(* IEC 61131-3 sources: ST-to-Python-Transpiler/AS Projekti/RampController/Program, 3 files *)

(* ---- Types.typ ---- *)
TYPE

END_TYPE

(* ---- Ramp.st ---- *)
PROGRAM _INIT
	(* Insert code here *)

END_PROGRAM

PROGRAM _CYCLIC
	(** --- RAMP CONTROLLER LOGIC --- **)
	Ramp(TARGET := UserSetpoint, CURRENT := CurrentValue, RAMP_UP := RampRateUp, RAMP_DOWN := RampRateDown, ENABLE := RampEnable, RESET := RampReset);
	SmoothSetpoint := Ramp.OUT;
	AtTarget := Ramp.REACHED;

	(** --- DEADBAND FILTER LOGIC --- **)
	Filter(IN := SensorRaw, DEADBAND := Deadband, CENTER := SmoothSetpoint);
	SensorFiltered := Filter.OUT;
	SensorActive := Filter.IS_ACTIVE;

END_PROGRAM

PROGRAM _EXIT
	(* Insert code here *)

END_PROGRAM

(* ---- Variables.var ---- *)
VAR
	UserSetpoint : REAL := 100.0;
	SensorRaw : REAL := 99.7;
	Ramp : RampController;
	Filter : DeadbandFilter; (** Control ramp behavior **)
	RampEnable : BOOL := TRUE;
	RampReset : BOOL := FALSE;
	RampRateUp : REAL := 1.0;
	RampRateDown : REAL := 2.0;
	CurrentValue : REAL := 90.0; (** Parameters for deadband filter **)
	Deadband : REAL := 0.5; (** Output: Ramped setpoint **)
	SmoothSetpoint : REAL; (** Output: Filtered sensor signal **)
	SensorFiltered : REAL; (** Output: TRUE when ramp reached target **)
	AtTarget : BOOL; (** Output: TRUE if sensor is outside deadband **)
	SensorActive : BOOL;
END_VAR
